Staubli VAL3: RecordJoint.pgx

public program RecordJoint(jointRx& x_jJDest, bool& x_bRes)
  local point l_pPoint
  local frame l_fFrame
begin

  link(l_fFrame,world)
  l_fFrame.trsf=TxtFile:fProduct.trsf*TxtFile:fTraj.trsf

  l_pPoint=here(TxtFile:tCfg,world)
  l_pPoint.trsf=l_pPoint.trsf*!TxtFile:fProduct.trsf*TxtFile:fPofffset.trsf*!TxtFile:fTraj.trsf
  l_pPoint.trsf=l_pPoint.trsf*!TxtFile:fToffset.trsf*!TxtFile:fArray.trsf
  link(l_pPoint,l_fFrame)
  x_jJDest=herej()
  x_bRes=pointToJoint(TxtFile:tCfg,x_jJDest,l_pPoint,x_jJDest)



end
